FUNCTION_BLOCK INTERNAL DefaultStringBuilder IMPLEMENTS StringBuilder, LimitedStringBuilder
VAR
  {attribute 'hide'}
  _workString : Tc2_System.T_MaxString;
END_VAR

METHOD PUBLIC Append : StringBuilder // Append text TO t current build STRING.
VAR_INPUT
  text : Tc2_System.T_MaxString; //text to append to current build string
END_VAR
_workString:= Tc2_Standard.CONCAT(_workString,text);
Append := THIS^;
END_METHOD

METHOD PUBLIC AppendIf : StringBuilder
VAR_INPUT
  condition : BOOL;
  text : Tc2_System.T_MaxString;
END_VAR
IF condition THEN
  _workString:= Tc2_Standard.CONCAT(_workString,text);
END_IF
AppendIf := THIS^;
END_METHOD

METHOD PUBLIC InsertAtLocation : StringBuilder
VAR_INPUT
  text : Tc2_System.T_MaxString;
  position : INT;
END_VAR
_workString := Tc2_Standard.INSERT(_workSTring,text,position);
InsertAtLocation  := THIS^;
END_METHOD

METHOD PadLeft : StringBuilder
VAR_INPUT
  text : Tc2_System.T_MaxString; // Text to append to current build string
  length : INT; // Total length of text + padding
  c : STRING(1); // Character to be padded left of text
END_VAR
VAR
  i : INT;
  padLength : INT;
END_VAR
// Add left padding
padLength := Tc2_Standard.LEN(text) - length;
FOR i := 1 TO padLength DO
  _workString:= Tc2_Standard.CONCAT(_workString, c);
END_FOR

// Add text
_workString:= Tc2_Standard.CONCAT(_workString,text);

PadLeft := THIS^;
END_METHOD

METHOD PUBLIC Reset : LimitedStringBuilder //Reset current build STRING TO an empty STRING.
_workString:='';
Reset := THIS^;
END_METHOD

METHOD PUBLIC ToString : Tc2_System.T_MaxString //Returns current build STRING.
ToString := _workString;
END_METHOD

END_FUNCTION_BLOCK

(* stored: Version 1.1.0.1
   POU DefaultStringBuilder: Id {62361e24-1326-47ec-af14-ad0e2274b160}, SpecialFunc None
   Method Append: Id {1435c08e-529b-4207-8673-c20f8fd97d5f}
   Method AppendIf: Id {10c3026e-ecd9-4569-8572-993e3a299766}
   Method InsertAtLocation: Id {5aa4c15e-8c20-4bcc-948c-bb970f0d1d01}
   Method PadLeft: Id {05b05d32-4814-42d9-8fdc-4f488852f39c}
   Method Reset: Id {270dbc93-3a82-4748-8588-b6dccf270a88}
   Method ToString: Id {e0c08440-9fdb-44a0-a847-5a6eb11ac8a7} *)
